{attribute 'qualified_only'}
{attribute 'strict'}
TYPE E_Enum :
(
	Member0 := 0,
	Member1,
	Member2
);
END_TYPE

(* stored: Version 1.1.0.1, ProductVersion 3.1.4024.4
   DUT E_Enum: Id {b6cdbd07-8b49-4a16-96cd-15e8ac69d4e9} *)
